// TIA Portal V18 export
// export: Created 2026-06-16T05:09:47.3581313Z, ExportSetting WithDefaults, DisplayName Totally Integrated Automation Portal, DisplayVersion V18 Update 5, DisplayName TIA Portal Openness, DisplayVersion V18 Update 5, DisplayName TIA Portal Version Control Interface, DisplayVersion V18, DisplayName SINAMICS Startdrive Advanced, DisplayVersion V18 SP2 Update 1, DisplayName SINAMICS Startdrive G110M, G120, G120C, G120D, G120P, G115D, DisplayVersion V18 SP2 Update 1, DisplayName SINAMICS Startdrive G130, G150, S120, S150, SINAMICS MV, S210, G220, S200, DisplayVersion V18 SP2 Update 1, DisplayName STEP 7 Professional, DisplayVersion V18 Update 5, DisplayName STEP 7 Safety, DisplayVersion V18, DisplayName WinCC Advanced / Unified PC, DisplayVersion V18 Update 5
FUNCTION "TEMPLATE--v1.0--04_ESTOP" : Void   // FC23, F_FBD
TITLE = SAFETY/EMERGENCY POWER CUT MANAGEMENT
{ S7_Optimized_Access := 'TRUE' }
VERSION : 0.1
// v1.0 First Emission
// stored: AutoNumber true, IsIECCheckEnabled false, UDAEnableTagReadback false
BEGIN

REGION Network 1: !!NetworkComment$$ Sorter, Doors<=4
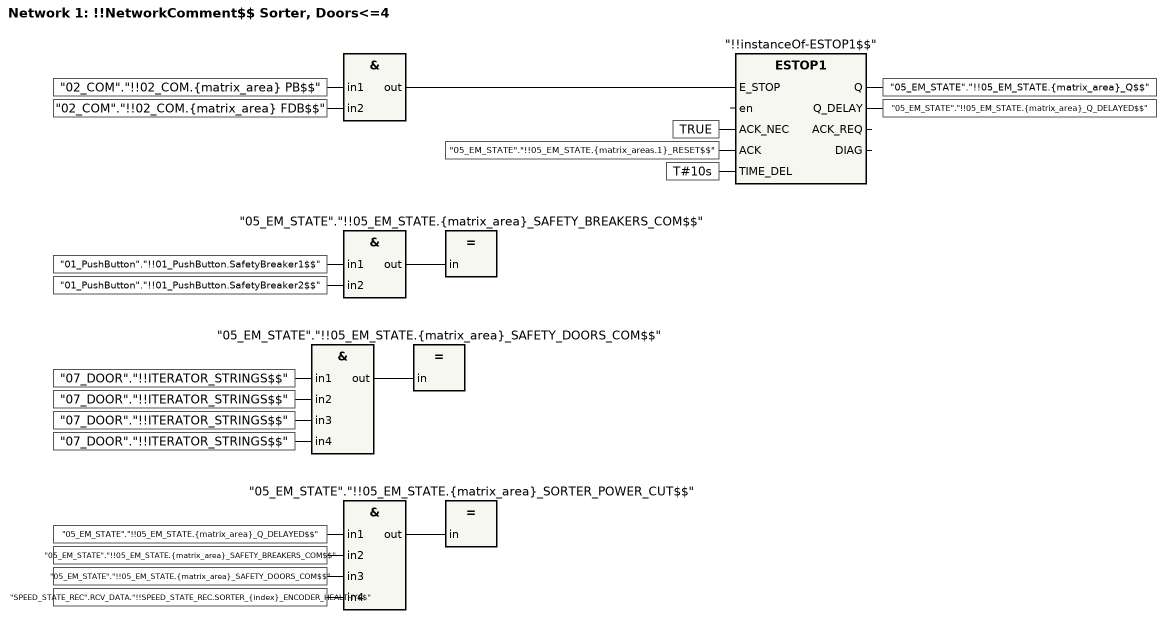
   "!!instanceOf-ESTOP1$$"(E_STOP := "02_COM"."!!02_COM.{matrix_area} PB$$" AND "02_COM"."!!02_COM.{matrix_area} FDB$$",   // ESTOP1
                           ACK_NEC := TRUE,
                           ACK := "05_EM_STATE"."!!05_EM_STATE.{matrix_areas.1}_RESET$$",
                           TIME_DEL := T#10s,
                           Q => "05_EM_STATE"."!!05_EM_STATE.{matrix_area}_Q$$",
                           Q_DELAY => "05_EM_STATE"."!!05_EM_STATE.{matrix_area}_Q_DELAYED$$");
   "05_EM_STATE"."!!05_EM_STATE.{matrix_area}_SAFETY_BREAKERS_COM$$" := "01_PushButton"."!!01_PushButton.SafetyBreaker1$$" AND "01_PushButton"."!!01_PushButton.SafetyBreaker2$$";
   "05_EM_STATE"."!!05_EM_STATE.{matrix_area}_SAFETY_DOORS_COM$$" := "07_DOOR"."!!ITERATOR_STRINGS$$" AND "07_DOOR"."!!ITERATOR_STRINGS$$" AND "07_DOOR"."!!ITERATOR_STRINGS$$" AND "07_DOOR"."!!ITERATOR_STRINGS$$";
   "05_EM_STATE"."!!05_EM_STATE.{matrix_area}_SORTER_POWER_CUT$$" := "05_EM_STATE"."!!05_EM_STATE.{matrix_area}_Q_DELAYED$$" AND "05_EM_STATE"."!!05_EM_STATE.{matrix_area}_SAFETY_BREAKERS_COM$$" AND "05_EM_STATE"."!!05_EM_STATE.{matrix_area}_SAFETY_DOORS_COM$$" AND "SPEED_STATE_REC".RCV_DATA."!!SPEED_STATE_REC.SORTER_{index}_ENCODER_HEALTHY$$";
END_REGION

REGION Network 2: !!NetworkComment$$ Sorter, Doors<=8
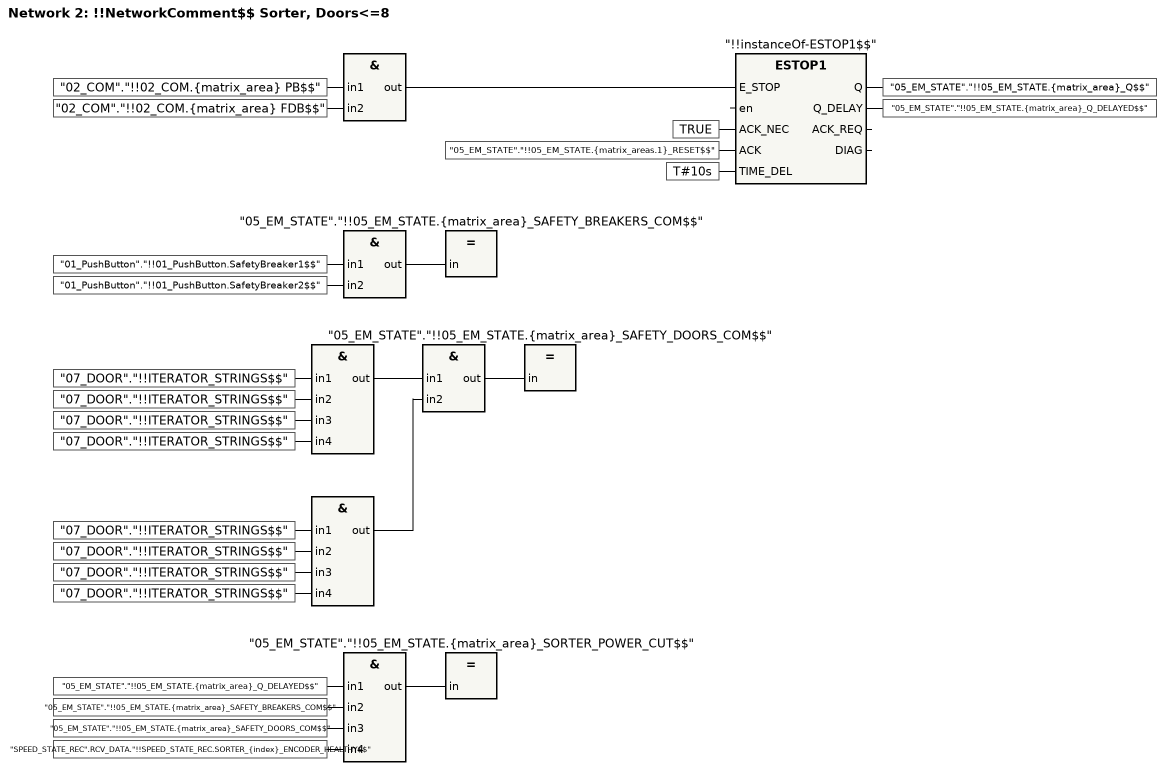
   "!!instanceOf-ESTOP1$$"(E_STOP := "02_COM"."!!02_COM.{matrix_area} PB$$" AND "02_COM"."!!02_COM.{matrix_area} FDB$$",   // ESTOP1
                           ACK_NEC := TRUE,
                           ACK := "05_EM_STATE"."!!05_EM_STATE.{matrix_areas.1}_RESET$$",
                           TIME_DEL := T#10s,
                           Q => "05_EM_STATE"."!!05_EM_STATE.{matrix_area}_Q$$",
                           Q_DELAY => "05_EM_STATE"."!!05_EM_STATE.{matrix_area}_Q_DELAYED$$");
   "05_EM_STATE"."!!05_EM_STATE.{matrix_area}_SAFETY_BREAKERS_COM$$" := "01_PushButton"."!!01_PushButton.SafetyBreaker1$$" AND "01_PushButton"."!!01_PushButton.SafetyBreaker2$$";
   "05_EM_STATE"."!!05_EM_STATE.{matrix_area}_SAFETY_DOORS_COM$$" := "07_DOOR"."!!ITERATOR_STRINGS$$" AND "07_DOOR"."!!ITERATOR_STRINGS$$" AND "07_DOOR"."!!ITERATOR_STRINGS$$" AND "07_DOOR"."!!ITERATOR_STRINGS$$" AND "07_DOOR"."!!ITERATOR_STRINGS$$" AND "07_DOOR"."!!ITERATOR_STRINGS$$" AND "07_DOOR"."!!ITERATOR_STRINGS$$" AND "07_DOOR"."!!ITERATOR_STRINGS$$";
   "05_EM_STATE"."!!05_EM_STATE.{matrix_area}_SORTER_POWER_CUT$$" := "05_EM_STATE"."!!05_EM_STATE.{matrix_area}_Q_DELAYED$$" AND "05_EM_STATE"."!!05_EM_STATE.{matrix_area}_SAFETY_BREAKERS_COM$$" AND "05_EM_STATE"."!!05_EM_STATE.{matrix_area}_SAFETY_DOORS_COM$$" AND "SPEED_STATE_REC".RCV_DATA."!!SPEED_STATE_REC.SORTER_{index}_ENCODER_HEALTHY$$";
END_REGION

REGION Network 3: !!NetworkComment$$ Sorter, Doors<=12
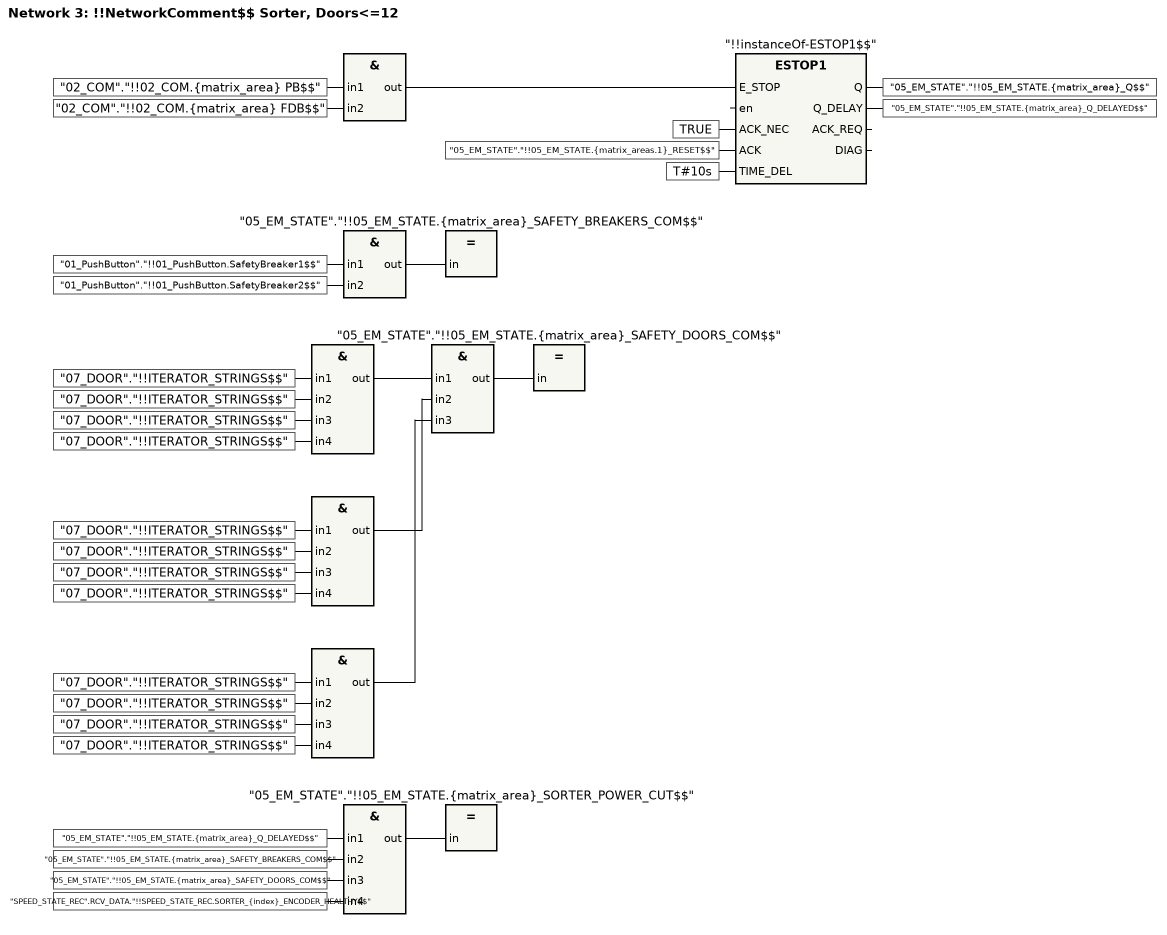
   "!!instanceOf-ESTOP1$$"(E_STOP := "02_COM"."!!02_COM.{matrix_area} PB$$" AND "02_COM"."!!02_COM.{matrix_area} FDB$$",   // ESTOP1
                           ACK_NEC := TRUE,
                           ACK := "05_EM_STATE"."!!05_EM_STATE.{matrix_areas.1}_RESET$$",
                           TIME_DEL := T#10s,
                           Q => "05_EM_STATE"."!!05_EM_STATE.{matrix_area}_Q$$",
                           Q_DELAY => "05_EM_STATE"."!!05_EM_STATE.{matrix_area}_Q_DELAYED$$");
   "05_EM_STATE"."!!05_EM_STATE.{matrix_area}_SAFETY_BREAKERS_COM$$" := "01_PushButton"."!!01_PushButton.SafetyBreaker1$$" AND "01_PushButton"."!!01_PushButton.SafetyBreaker2$$";
   "05_EM_STATE"."!!05_EM_STATE.{matrix_area}_SAFETY_DOORS_COM$$" := "07_DOOR"."!!ITERATOR_STRINGS$$" AND "07_DOOR"."!!ITERATOR_STRINGS$$" AND "07_DOOR"."!!ITERATOR_STRINGS$$" AND "07_DOOR"."!!ITERATOR_STRINGS$$" AND "07_DOOR"."!!ITERATOR_STRINGS$$" AND "07_DOOR"."!!ITERATOR_STRINGS$$" AND "07_DOOR"."!!ITERATOR_STRINGS$$" AND "07_DOOR"."!!ITERATOR_STRINGS$$" AND "07_DOOR"."!!ITERATOR_STRINGS$$" AND "07_DOOR"."!!ITERATOR_STRINGS$$" AND "07_DOOR"."!!ITERATOR_STRINGS$$" AND "07_DOOR"."!!ITERATOR_STRINGS$$";
   "05_EM_STATE"."!!05_EM_STATE.{matrix_area}_SORTER_POWER_CUT$$" := "05_EM_STATE"."!!05_EM_STATE.{matrix_area}_Q_DELAYED$$" AND "05_EM_STATE"."!!05_EM_STATE.{matrix_area}_SAFETY_BREAKERS_COM$$" AND "05_EM_STATE"."!!05_EM_STATE.{matrix_area}_SAFETY_DOORS_COM$$" AND "SPEED_STATE_REC".RCV_DATA."!!SPEED_STATE_REC.SORTER_{index}_ENCODER_HEALTHY$$";
END_REGION

REGION Network 4: !!NetworkComment$$ Sorter, Doors<=16
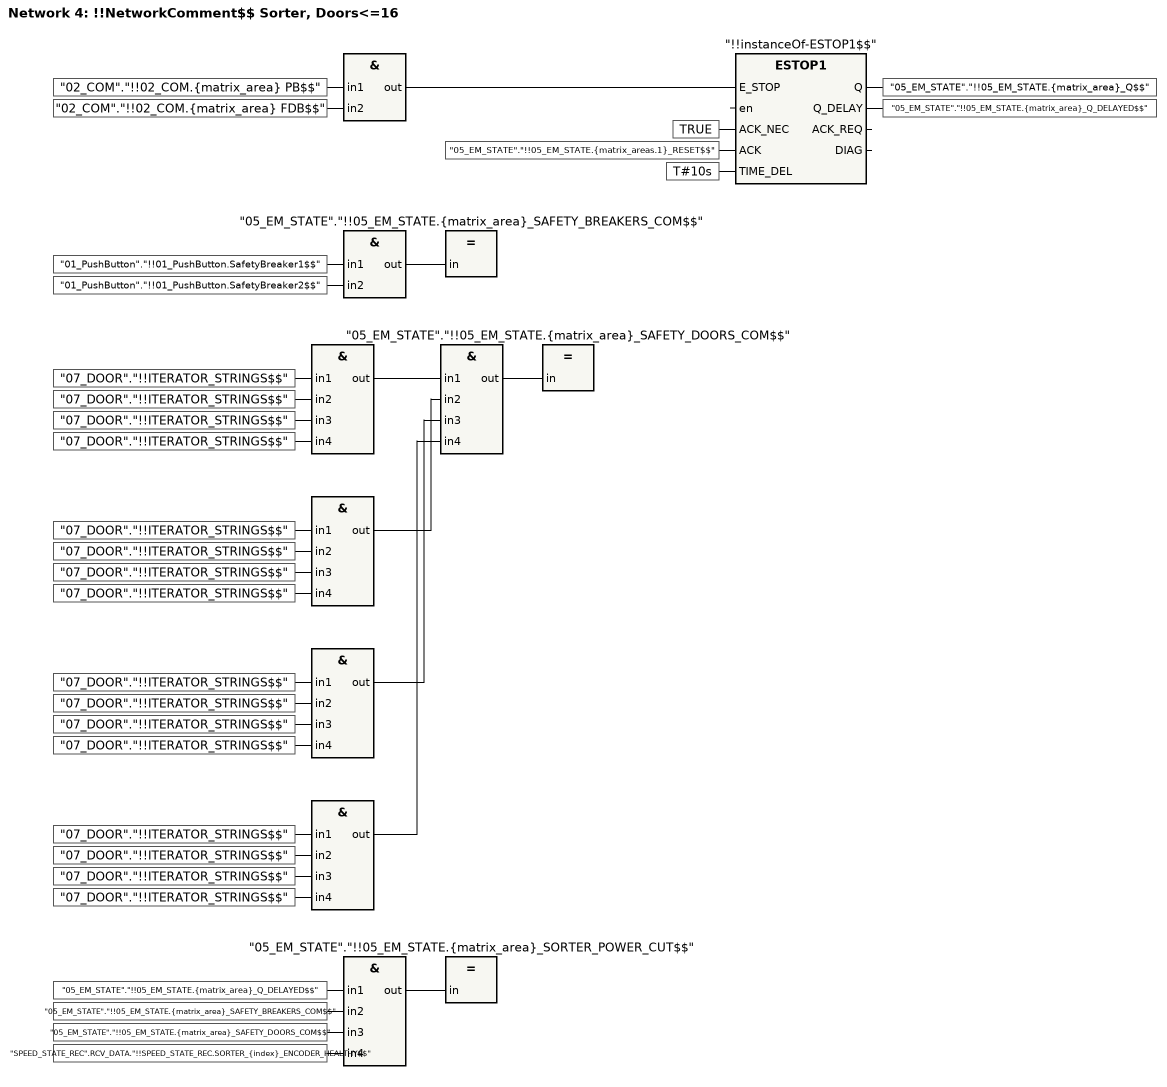
   "!!instanceOf-ESTOP1$$"(E_STOP := "02_COM"."!!02_COM.{matrix_area} PB$$" AND "02_COM"."!!02_COM.{matrix_area} FDB$$",   // ESTOP1
                           ACK_NEC := TRUE,
                           ACK := "05_EM_STATE"."!!05_EM_STATE.{matrix_areas.1}_RESET$$",
                           TIME_DEL := T#10s,
                           Q => "05_EM_STATE"."!!05_EM_STATE.{matrix_area}_Q$$",
                           Q_DELAY => "05_EM_STATE"."!!05_EM_STATE.{matrix_area}_Q_DELAYED$$");
   "05_EM_STATE"."!!05_EM_STATE.{matrix_area}_SAFETY_BREAKERS_COM$$" := "01_PushButton"."!!01_PushButton.SafetyBreaker1$$" AND "01_PushButton"."!!01_PushButton.SafetyBreaker2$$";
   "05_EM_STATE"."!!05_EM_STATE.{matrix_area}_SAFETY_DOORS_COM$$" := "07_DOOR"."!!ITERATOR_STRINGS$$" AND "07_DOOR"."!!ITERATOR_STRINGS$$" AND "07_DOOR"."!!ITERATOR_STRINGS$$" AND "07_DOOR"."!!ITERATOR_STRINGS$$" AND "07_DOOR"."!!ITERATOR_STRINGS$$" AND "07_DOOR"."!!ITERATOR_STRINGS$$" AND "07_DOOR"."!!ITERATOR_STRINGS$$" AND "07_DOOR"."!!ITERATOR_STRINGS$$" AND "07_DOOR"."!!ITERATOR_STRINGS$$" AND "07_DOOR"."!!ITERATOR_STRINGS$$" AND "07_DOOR"."!!ITERATOR_STRINGS$$" AND "07_DOOR"."!!ITERATOR_STRINGS$$" AND "07_DOOR"."!!ITERATOR_STRINGS$$" AND "07_DOOR"."!!ITERATOR_STRINGS$$" AND "07_DOOR"."!!ITERATOR_STRINGS$$" AND "07_DOOR"."!!ITERATOR_STRINGS$$";
   "05_EM_STATE"."!!05_EM_STATE.{matrix_area}_SORTER_POWER_CUT$$" := "05_EM_STATE"."!!05_EM_STATE.{matrix_area}_Q_DELAYED$$" AND "05_EM_STATE"."!!05_EM_STATE.{matrix_area}_SAFETY_BREAKERS_COM$$" AND "05_EM_STATE"."!!05_EM_STATE.{matrix_area}_SAFETY_DOORS_COM$$" AND "SPEED_STATE_REC".RCV_DATA."!!SPEED_STATE_REC.SORTER_{index}_ENCODER_HEALTHY$$";
END_REGION

REGION Network 5: !!NetworkComment$$ Sorter, Doors<=20
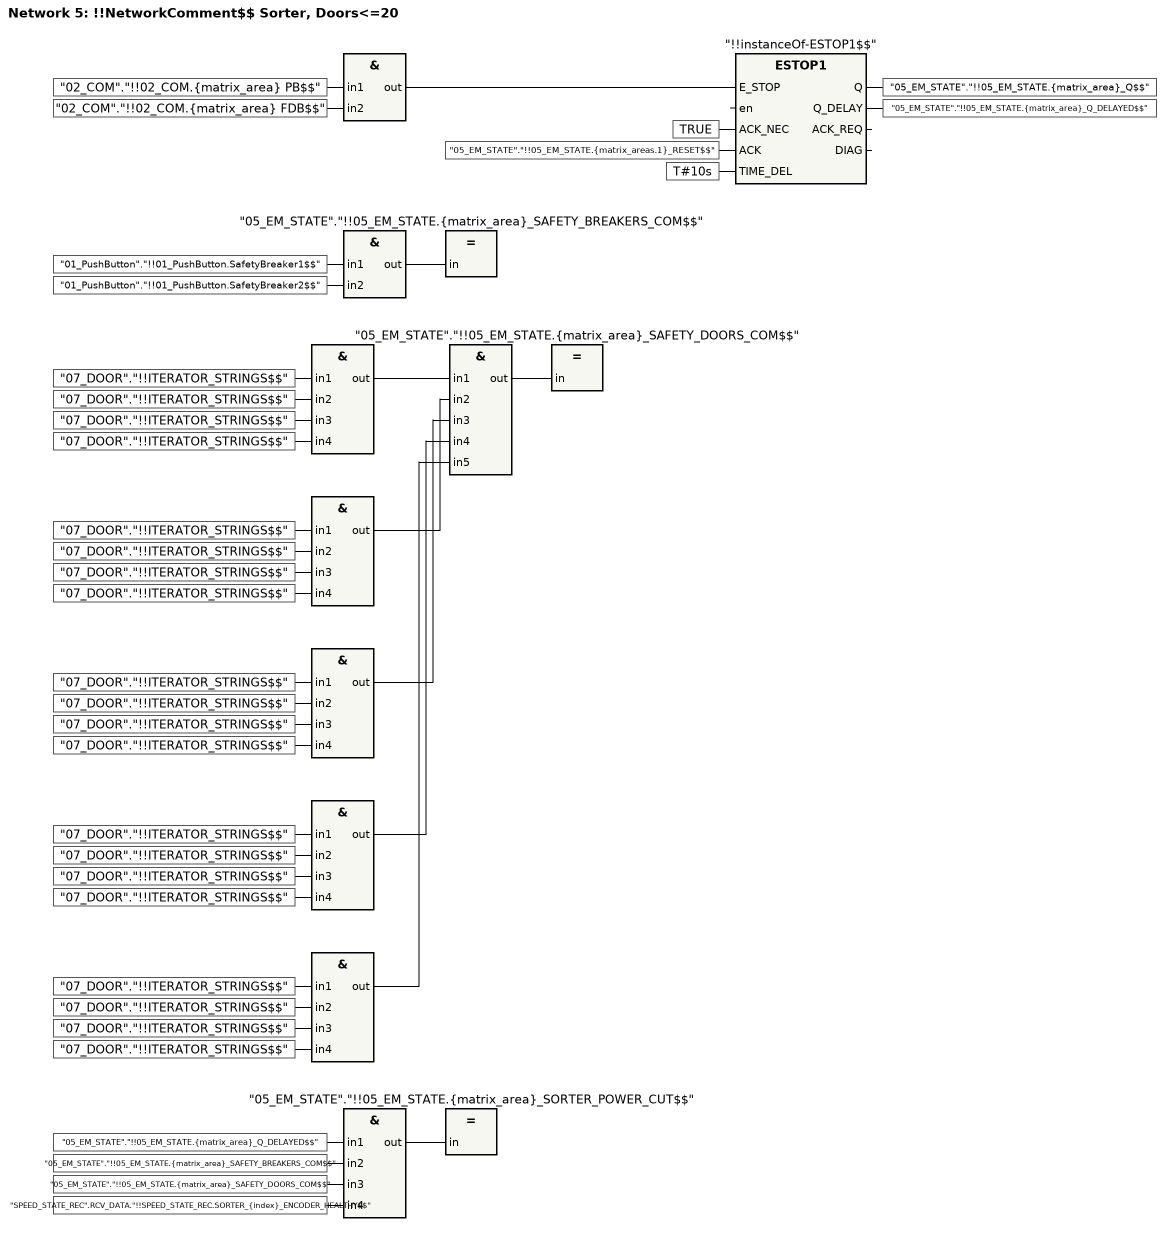
   "!!instanceOf-ESTOP1$$"(E_STOP := "02_COM"."!!02_COM.{matrix_area} PB$$" AND "02_COM"."!!02_COM.{matrix_area} FDB$$",   // ESTOP1
                           ACK_NEC := TRUE,
                           ACK := "05_EM_STATE"."!!05_EM_STATE.{matrix_areas.1}_RESET$$",
                           TIME_DEL := T#10s,
                           Q => "05_EM_STATE"."!!05_EM_STATE.{matrix_area}_Q$$",
                           Q_DELAY => "05_EM_STATE"."!!05_EM_STATE.{matrix_area}_Q_DELAYED$$");
   "05_EM_STATE"."!!05_EM_STATE.{matrix_area}_SAFETY_BREAKERS_COM$$" := "01_PushButton"."!!01_PushButton.SafetyBreaker1$$" AND "01_PushButton"."!!01_PushButton.SafetyBreaker2$$";
   "05_EM_STATE"."!!05_EM_STATE.{matrix_area}_SAFETY_DOORS_COM$$" := "07_DOOR"."!!ITERATOR_STRINGS$$" AND "07_DOOR"."!!ITERATOR_STRINGS$$" AND "07_DOOR"."!!ITERATOR_STRINGS$$" AND "07_DOOR"."!!ITERATOR_STRINGS$$" AND "07_DOOR"."!!ITERATOR_STRINGS$$" AND "07_DOOR"."!!ITERATOR_STRINGS$$" AND "07_DOOR"."!!ITERATOR_STRINGS$$" AND "07_DOOR"."!!ITERATOR_STRINGS$$" AND "07_DOOR"."!!ITERATOR_STRINGS$$" AND "07_DOOR"."!!ITERATOR_STRINGS$$" AND "07_DOOR"."!!ITERATOR_STRINGS$$" AND "07_DOOR"."!!ITERATOR_STRINGS$$" AND "07_DOOR"."!!ITERATOR_STRINGS$$" AND "07_DOOR"."!!ITERATOR_STRINGS$$" AND "07_DOOR"."!!ITERATOR_STRINGS$$" AND "07_DOOR"."!!ITERATOR_STRINGS$$" AND "07_DOOR"."!!ITERATOR_STRINGS$$" AND "07_DOOR"."!!ITERATOR_STRINGS$$" AND "07_DOOR"."!!ITERATOR_STRINGS$$" AND "07_DOOR"."!!ITERATOR_STRINGS$$";
   "05_EM_STATE"."!!05_EM_STATE.{matrix_area}_SORTER_POWER_CUT$$" := "05_EM_STATE"."!!05_EM_STATE.{matrix_area}_Q_DELAYED$$" AND "05_EM_STATE"."!!05_EM_STATE.{matrix_area}_SAFETY_BREAKERS_COM$$" AND "05_EM_STATE"."!!05_EM_STATE.{matrix_area}_SAFETY_DOORS_COM$$" AND "SPEED_STATE_REC".RCV_DATA."!!SPEED_STATE_REC.SORTER_{index}_ENCODER_HEALTHY$$";
END_REGION

REGION Network 6: !!NetworkComment$$ Conveyors / Other Machines, Acknowledge Required
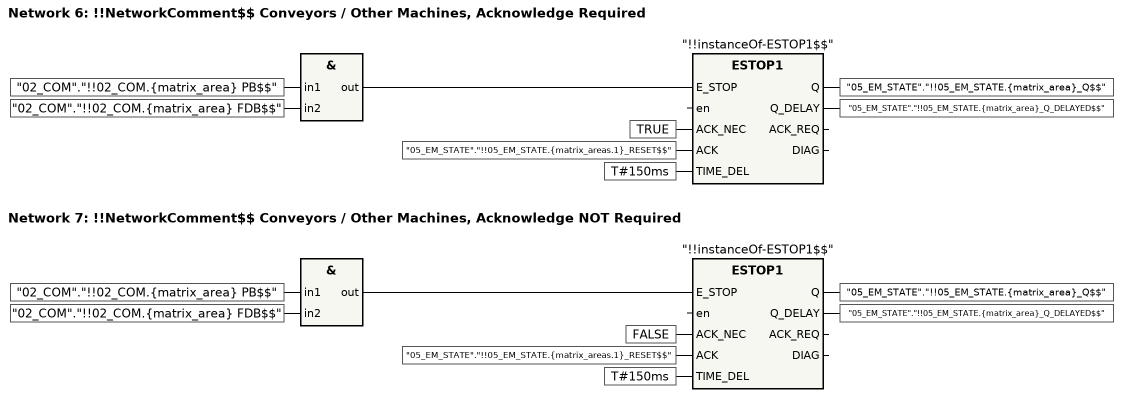
   "!!instanceOf-ESTOP1$$"(E_STOP := "02_COM"."!!02_COM.{matrix_area} PB$$" AND "02_COM"."!!02_COM.{matrix_area} FDB$$",   // ESTOP1
                           ACK_NEC := TRUE,
                           ACK := "05_EM_STATE"."!!05_EM_STATE.{matrix_areas.1}_RESET$$",
                           TIME_DEL := T#150ms,
                           Q => "05_EM_STATE"."!!05_EM_STATE.{matrix_area}_Q$$",
                           Q_DELAY => "05_EM_STATE"."!!05_EM_STATE.{matrix_area}_Q_DELAYED$$");
END_REGION

REGION Network 7: !!NetworkComment$$ Conveyors / Other Machines, Acknowledge NOT Required
   "!!instanceOf-ESTOP1$$"(E_STOP := "02_COM"."!!02_COM.{matrix_area} PB$$" AND "02_COM"."!!02_COM.{matrix_area} FDB$$",   // ESTOP1
                           ACK_NEC := FALSE,
                           ACK := "05_EM_STATE"."!!05_EM_STATE.{matrix_areas.1}_RESET$$",
                           TIME_DEL := T#150ms,
                           Q => "05_EM_STATE"."!!05_EM_STATE.{matrix_area}_Q$$",
                           Q_DELAY => "05_EM_STATE"."!!05_EM_STATE.{matrix_area}_Q_DELAYED$$");
END_REGION
END_FUNCTION
